FUNCTION_BLOCK OffsetDecorator IMPLEMENTS ITF_Analogue
VAR
	wrappee : ITF_Analogue;
	UpperLimit: BOOL;
END_VAR

METHOD GetValue : lreal
IF (THIS^.wrappee <> 0) THEN
 	GetValue := THIS^.wrappee.GetValue() - 10.0;
END_IF
END_METHOD

END_FUNCTION_BLOCK

(* stored: Version 1.1.0.1, ProductVersion 3.1.4024.12
   POU OffsetDecorator: Id {9de537f0-d915-4a60-874f-abd46092d676}, SpecialFunc None
   Method GetValue: Id {d38bb00c-731a-4c41-89cb-c327be740ea4} *)
